FUNCTION_BLOCK FB_010_ReadRParameter

VAR_INPUT
	Execute:BOOL;
    fbnChannelid:UDINT;	
END_VAR
VAR_OUTPUT
	nRParamAry:ARRAY[0..19] OF LREAL;
END_VAR
VAR
	fbReadRParams:ItpReadRParams;
END_VAR



	fbReadRParams(
	bExecute:= Execute, 
	nChnId:= fbnChannelid, 
	pAddr:= ADR(nRParamAry), 
	nIndex:= 0, 
	nCount:= 20, 
	tTimeOut:= T#2S, 
	bBusy=> , 
	bErr=> , 
	nErrId=> );

END_FUNCTION_BLOCK

(* stored: Version 1.1.0.1, ProductVersion 3.1.4024.12
   POU FB_010_ReadRParameter: Id {cf7204ed-bfd9-446c-b4f0-645a278d579e}, SpecialFunc None *)
